{attribute 'qualified_only'}
{attribute 'strict'}
{attribute 'to_string'}
TYPE INTERSECTION_TRAFFIC_LIGHTS_STATE :
(
	ALL_OFF := 0,
	ALL_YELLOW,
	_1_3_GREEN_AND_2_4_RED,
	_1_3_YELLOW_AND_2_4_YELLOW,
	_2_4_GREEN_AND_1_3_RED,
	_2_4_YELLOW_AND_1_3_YELLOW
);
END_TYPE

(* stored: Version 1.1.0.1
   DUT INTERSECTION_TRAFFIC_LIGHTS_STATE: Id {d3aa784f-61dc-4dcb-9bf6-937a3bff250b} *)
